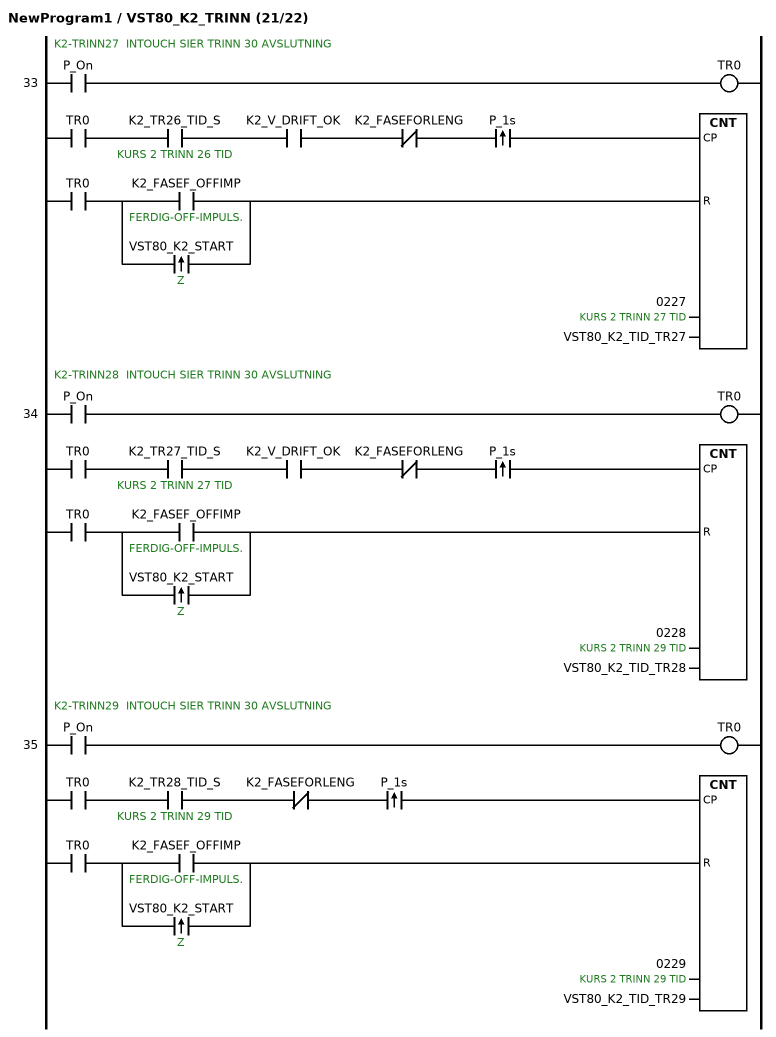
; [picture p216: NewProgram1 / VST80_K2_TRINN, rungs 33-35]
; rung 33: K2-TRINN27  INTOUCH SIER TRINN 30 AVSLUTNING
LD P_On
OUT TR0
AND K2_TR26_TID_S  ; KURS 2 TRINN 26 TID
AND K2_V_DRIFT_OK
ANDNOT K2_FASEFORLENG
@AND P_1s
LD TR0
LD K2_FASEF_OFFIMP  ; FERDIG-OFF-IMPULS.
@OR VST80_K2_START  ; Z
ANDLD
CNT 0227 VST80_K2_TID_TR27  ; KURS 2 TRINN 27 TID
; rung 34: K2-TRINN28  INTOUCH SIER TRINN 30 AVSLUTNING
LD P_On
OUT TR0
AND K2_TR27_TID_S  ; KURS 2 TRINN 27 TID
AND K2_V_DRIFT_OK
ANDNOT K2_FASEFORLENG
@AND P_1s
LD TR0
LD K2_FASEF_OFFIMP  ; FERDIG-OFF-IMPULS.
@OR VST80_K2_START  ; Z
ANDLD
CNT 0228 VST80_K2_TID_TR28  ; KURS 2 TRINN 29 TID
; rung 35: K2-TRINN29  INTOUCH SIER TRINN 30 AVSLUTNING
LD P_On
OUT TR0
AND K2_TR28_TID_S  ; KURS 2 TRINN 29 TID
ANDNOT K2_FASEFORLENG
@AND P_1s
LD TR0
LD K2_FASEF_OFFIMP  ; FERDIG-OFF-IMPULS.
@OR VST80_K2_START  ; Z
ANDLD
CNT 0229 VST80_K2_TID_TR29  ; KURS 2 TRINN 29 TID

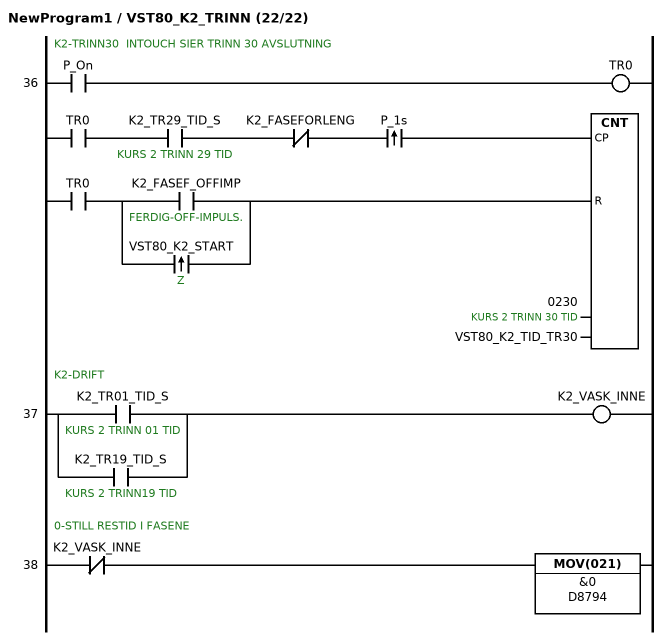
; rung 36: K2-TRINN30  INTOUCH SIER TRINN 30 AVSLUTNING
LD P_On
OUT TR0
AND K2_TR29_TID_S  ; KURS 2 TRINN 29 TID
ANDNOT K2_FASEFORLENG
@AND P_1s
LD TR0
LD K2_FASEF_OFFIMP  ; FERDIG-OFF-IMPULS.
@OR VST80_K2_START  ; Z
ANDLD
CNT 0230 VST80_K2_TID_TR30  ; KURS 2 TRINN 30 TID
; rung 37: K2-DRIFT
LD K2_TR01_TID_S  ; KURS 2 TRINN 01 TID
OR K2_TR19_TID_S  ; KURS 2 TRINN19 TID
OUT K2_VASK_INNE
; rung 38: 0-STILL RESTID I FASENE
LDNOT K2_VASK_INNE
MOV(021) &0 D8794

### Section VST80_K2_ANALOGSIGN_INN

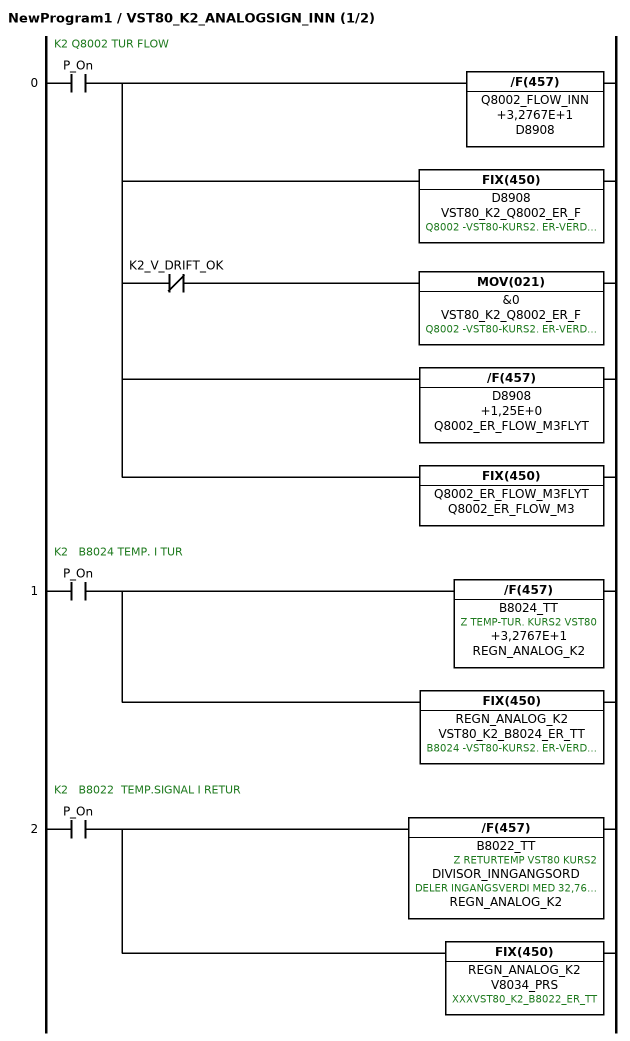
; rung 0: K2 Q8002 TUR FLOW
LD P_On
OUT TR0
/F(457) Q8002_FLOW_INN +3,2767E+1 D8908
FIX(450) D8908 VST80_K2_Q8002_ER_F  ; Q8002 -VST80-KURS2. ER-VERDI FLOW I TUR
ANDNOT K2_V_DRIFT_OK
MOV(021) &0 VST80_K2_Q8002_ER_F  ; Q8002 -VST80-KURS2. ER-VERDI FLOW I TUR
LD TR0
/F(457) D8908 +1,25E+0 Q8002_ER_FLOW_M3FLYT
FIX(450) Q8002_ER_FLOW_M3FLYT Q8002_ER_FLOW_M3
; rung 1: K2   B8024 TEMP. I TUR
LD P_On
/F(457) B8024_TT +3,2767E+1 REGN_ANALOG_K2  ; Z TEMP-TUR. KURS2 VST80
FIX(450) REGN_ANALOG_K2 VST80_K2_B8024_ER_TT  ; B8024 -VST80-KURS2. ER-VERDI TEMPERATUR I TUR TIL VST
; rung 2: K2   B8022  TEMP.SIGNAL I RETUR
LD P_On
/F(457) B8022_TT DIVISOR_INNGANGSORD REGN_ANALOG_K2  ; Z RETURTEMP VST80 KURS2, DELER INGANGSVERDI MED 32,760 FOR OMREGNING TIL 0-1000
FIX(450) REGN_ANALOG_K2 V8034_PRS  ; XXXVST80_K2_B8022_ER_TT

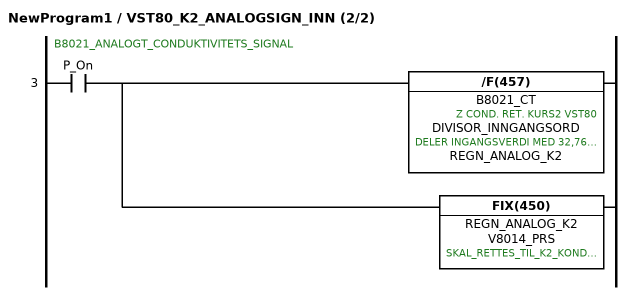
; rung 3: B8021_ANALOGT_CONDUKTIVITETS_SIGNAL
LD P_On
/F(457) B8021_CT DIVISOR_INNGANGSORD REGN_ANALOG_K2  ; Z COND. RET. KURS2 VST80, DELER INGANGSVERDI MED 32,760 FOR OMREGNING TIL 0-1000
FIX(450) REGN_ANALOG_K2 V8014_PRS  ; SKAL_RETTES_TIL_K2_KOND_ERVERDI

### Section VST_80_K2_TYPE_VASK
; KOMMANDOGIVNING FOR VALG AV TYPE VASK. / 2: DESINFEKSJON / 3: FORSKYLL

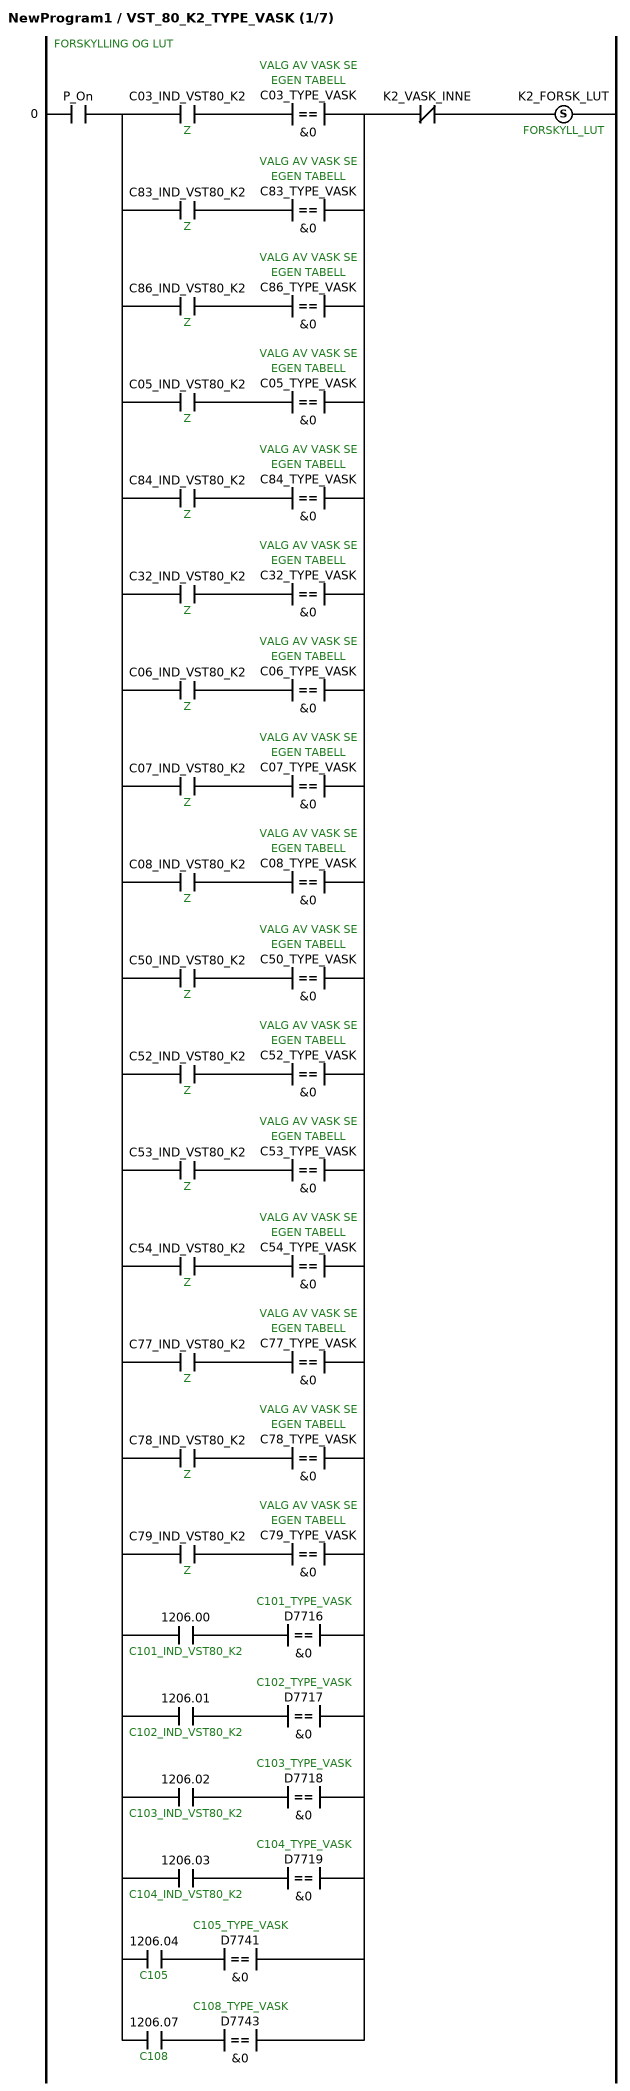
; rung 0: FORSKYLLING OG LUT
LD P_On
LD C03_IND_VST80_K2  ; Z
AND=(300) C03_TYPE_VASK &0  ; VALG AV VASK SE EGEN TABELL
LD C83_IND_VST80_K2  ; Z
AND=(300) C83_TYPE_VASK &0  ; VALG AV VASK SE EGEN TABELL
ORLD
LD C86_IND_VST80_K2  ; Z
AND=(300) C86_TYPE_VASK &0  ; VALG AV VASK SE EGEN TABELL
ORLD
LD C05_IND_VST80_K2  ; Z
AND=(300) C05_TYPE_VASK &0  ; VALG AV VASK SE EGEN TABELL
ORLD
LD C84_IND_VST80_K2  ; Z
AND=(300) C84_TYPE_VASK &0  ; VALG AV VASK SE EGEN TABELL
ORLD
LD C32_IND_VST80_K2  ; Z
AND=(300) C32_TYPE_VASK &0  ; VALG AV VASK SE EGEN TABELL
ORLD
LD C06_IND_VST80_K2  ; Z
AND=(300) C06_TYPE_VASK &0  ; VALG AV VASK SE EGEN TABELL
ORLD
LD C07_IND_VST80_K2  ; Z
AND=(300) C07_TYPE_VASK &0  ; VALG AV VASK SE EGEN TABELL
ORLD
LD C08_IND_VST80_K2  ; Z
AND=(300) C08_TYPE_VASK &0  ; VALG AV VASK SE EGEN TABELL
ORLD
LD C50_IND_VST80_K2  ; Z
AND=(300) C50_TYPE_VASK &0  ; VALG AV VASK SE EGEN TABELL
ORLD
LD C52_IND_VST80_K2  ; Z
AND=(300) C52_TYPE_VASK &0  ; VALG AV VASK SE EGEN TABELL
ORLD
LD C53_IND_VST80_K2  ; Z
AND=(300) C53_TYPE_VASK &0  ; VALG AV VASK SE EGEN TABELL
ORLD
LD C54_IND_VST80_K2  ; Z
AND=(300) C54_TYPE_VASK &0  ; VALG AV VASK SE EGEN TABELL
ORLD
LD C77_IND_VST80_K2  ; Z
AND=(300) C77_TYPE_VASK &0  ; VALG AV VASK SE EGEN TABELL
ORLD
LD C78_IND_VST80_K2  ; Z
AND=(300) C78_TYPE_VASK &0  ; VALG AV VASK SE EGEN TABELL
ORLD
LD C79_IND_VST80_K2  ; Z
AND=(300) C79_TYPE_VASK &0  ; VALG AV VASK SE EGEN TABELL
ORLD
LD 1206.00  ; C101_IND_VST80_K2
AND=(300) D7716 &0  ; C101_TYPE_VASK
ORLD
LD 1206.01  ; C102_IND_VST80_K2
AND=(300) D7717 &0  ; C102_TYPE_VASK
ORLD
LD 1206.02  ; C103_IND_VST80_K2
AND=(300) D7718 &0  ; C103_TYPE_VASK
ORLD
LD 1206.03  ; C104_IND_VST80_K2
AND=(300) D7719 &0  ; C104_TYPE_VASK
ORLD
LD 1206.04  ; C105
AND=(300) D7741 &0  ; C105_TYPE_VASK
ORLD
LD 1206.07  ; C108
AND=(300) D7743 &0  ; C108_TYPE_VASK
ORLD
ANDLD
ANDNOT K2_VASK_INNE
SET K2_FORSK_LUT  ; FORSKYLL_LUT

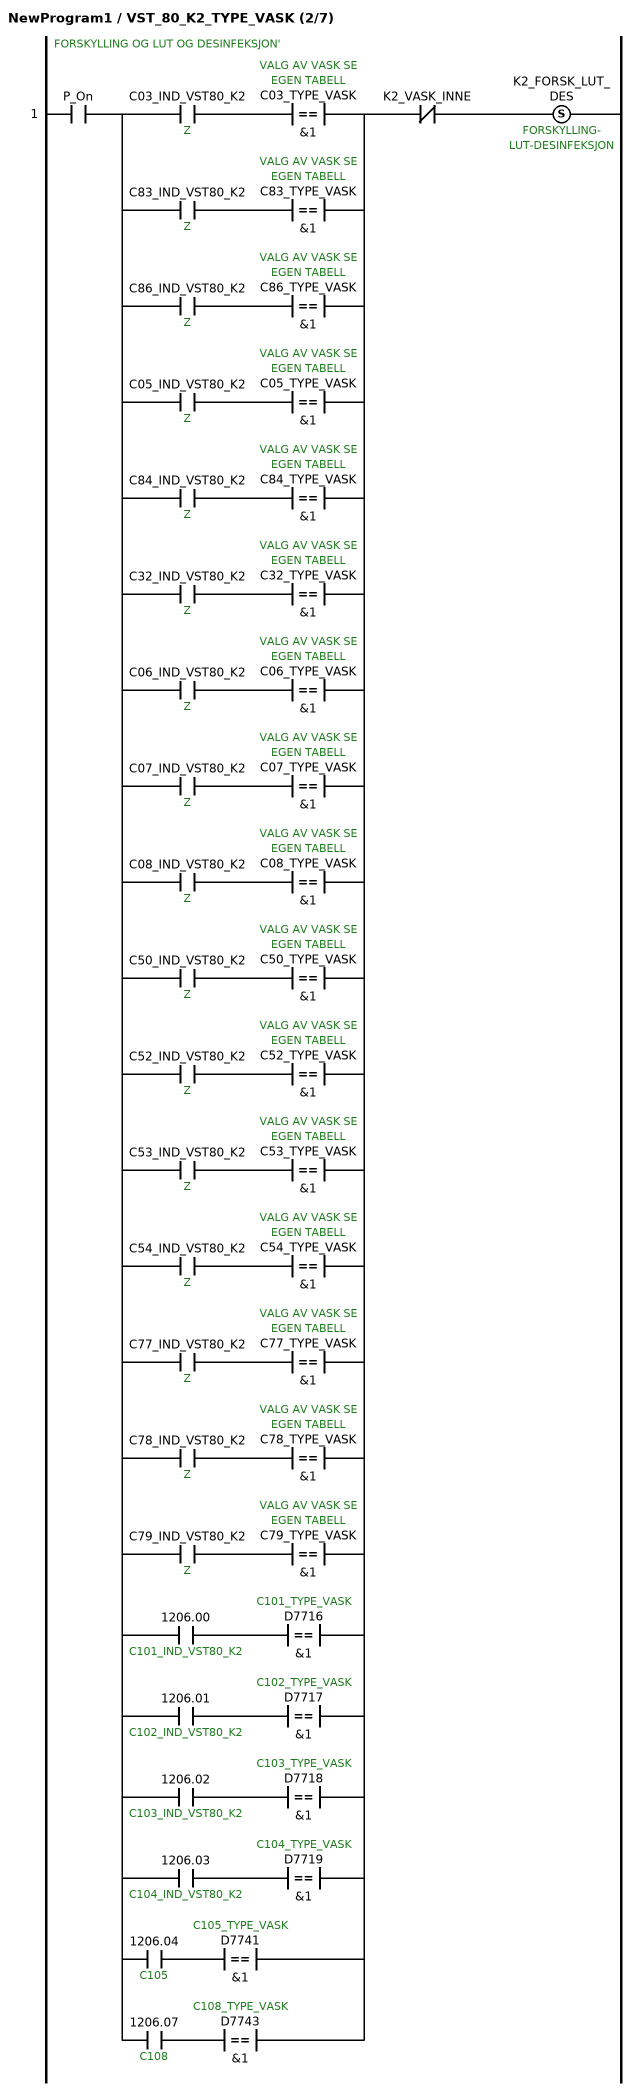
; rung 1: FORSKYLLING OG LUT OG DESINFEKSJON'
LD P_On
LD C03_IND_VST80_K2  ; Z
AND=(300) C03_TYPE_VASK &1  ; VALG AV VASK SE EGEN TABELL
LD C83_IND_VST80_K2  ; Z
AND=(300) C83_TYPE_VASK &1  ; VALG AV VASK SE EGEN TABELL
ORLD
LD C86_IND_VST80_K2  ; Z
AND=(300) C86_TYPE_VASK &1  ; VALG AV VASK SE EGEN TABELL
ORLD
LD C05_IND_VST80_K2  ; Z
AND=(300) C05_TYPE_VASK &1  ; VALG AV VASK SE EGEN TABELL
ORLD
LD C84_IND_VST80_K2  ; Z
AND=(300) C84_TYPE_VASK &1  ; VALG AV VASK SE EGEN TABELL
ORLD
LD C32_IND_VST80_K2  ; Z
AND=(300) C32_TYPE_VASK &1  ; VALG AV VASK SE EGEN TABELL
ORLD
LD C06_IND_VST80_K2  ; Z
AND=(300) C06_TYPE_VASK &1  ; VALG AV VASK SE EGEN TABELL
ORLD
LD C07_IND_VST80_K2  ; Z
AND=(300) C07_TYPE_VASK &1  ; VALG AV VASK SE EGEN TABELL
ORLD
LD C08_IND_VST80_K2  ; Z
AND=(300) C08_TYPE_VASK &1  ; VALG AV VASK SE EGEN TABELL
ORLD
LD C50_IND_VST80_K2  ; Z
AND=(300) C50_TYPE_VASK &1  ; VALG AV VASK SE EGEN TABELL
ORLD
LD C52_IND_VST80_K2  ; Z
AND=(300) C52_TYPE_VASK &1  ; VALG AV VASK SE EGEN TABELL
ORLD
LD C53_IND_VST80_K2  ; Z
AND=(300) C53_TYPE_VASK &1  ; VALG AV VASK SE EGEN TABELL
ORLD
LD C54_IND_VST80_K2  ; Z
AND=(300) C54_TYPE_VASK &1  ; VALG AV VASK SE EGEN TABELL
ORLD
LD C77_IND_VST80_K2  ; Z
AND=(300) C77_TYPE_VASK &1  ; VALG AV VASK SE EGEN TABELL
ORLD
LD C78_IND_VST80_K2  ; Z
AND=(300) C78_TYPE_VASK &1  ; VALG AV VASK SE EGEN TABELL
ORLD
LD C79_IND_VST80_K2  ; Z
AND=(300) C79_TYPE_VASK &1  ; VALG AV VASK SE EGEN TABELL
ORLD
LD 1206.00  ; C101_IND_VST80_K2
AND=(300) D7716 &1  ; C101_TYPE_VASK
ORLD
LD 1206.01  ; C102_IND_VST80_K2
AND=(300) D7717 &1  ; C102_TYPE_VASK
ORLD
LD 1206.02  ; C103_IND_VST80_K2
AND=(300) D7718 &1  ; C103_TYPE_VASK
ORLD
LD 1206.03  ; C104_IND_VST80_K2
AND=(300) D7719 &1  ; C104_TYPE_VASK
ORLD
LD 1206.04  ; C105
AND=(300) D7741 &1  ; C105_TYPE_VASK
ORLD
LD 1206.07  ; C108
AND=(300) D7743 &1  ; C108_TYPE_VASK
ORLD
ANDLD
ANDNOT K2_VASK_INNE
SET K2_FORSK_LUT_DES  ; FORSKYLLING- LUT-DESINFEKSJON

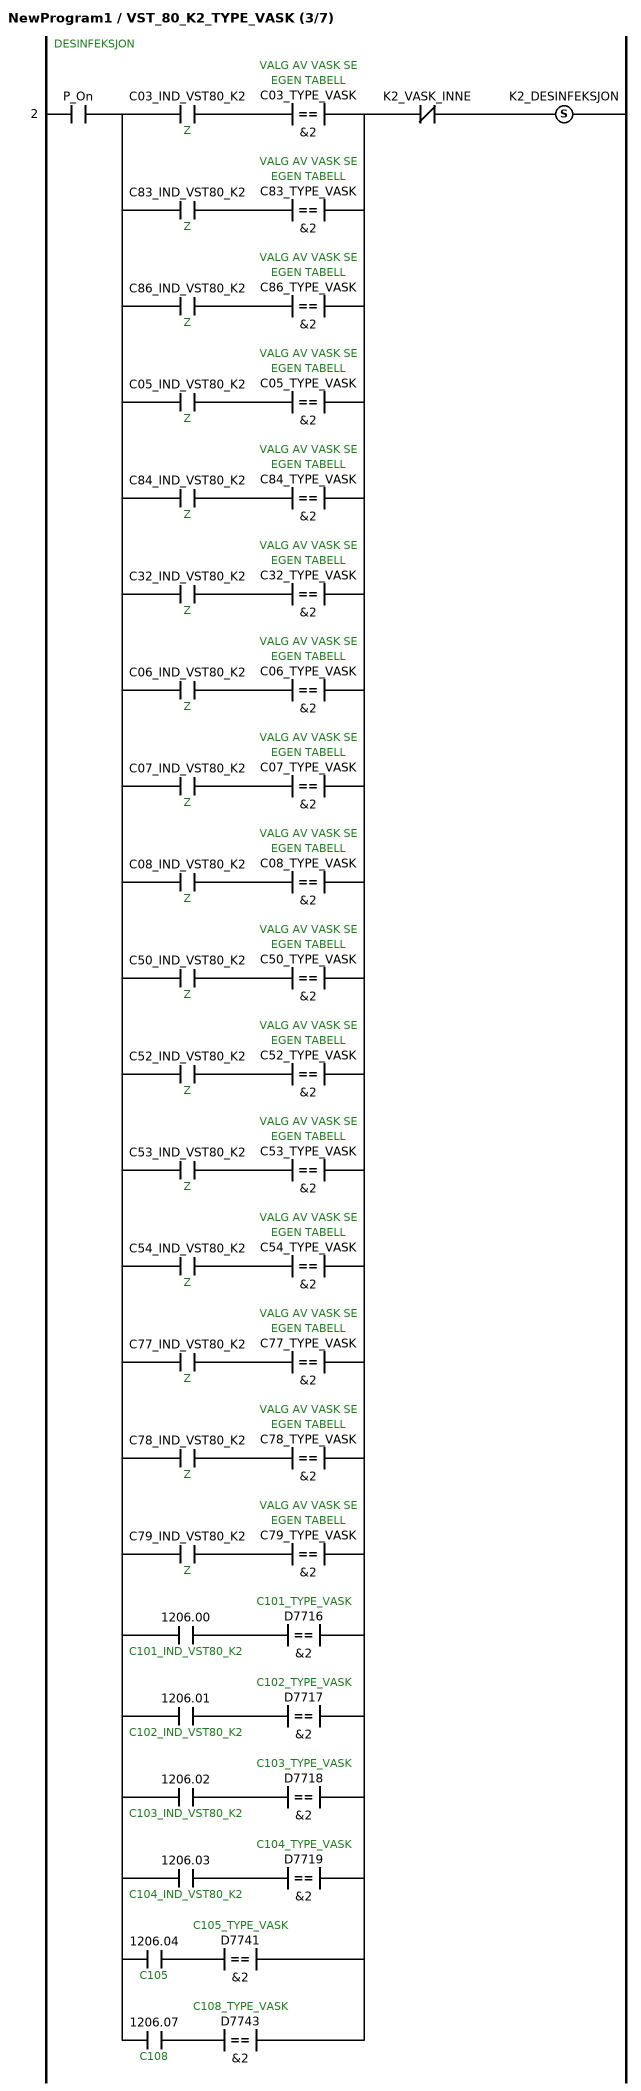
; rung 2: DESINFEKSJON
LD P_On
LD C03_IND_VST80_K2  ; Z
AND=(300) C03_TYPE_VASK &2  ; VALG AV VASK SE EGEN TABELL
LD C83_IND_VST80_K2  ; Z
AND=(300) C83_TYPE_VASK &2  ; VALG AV VASK SE EGEN TABELL
ORLD
LD C86_IND_VST80_K2  ; Z
AND=(300) C86_TYPE_VASK &2  ; VALG AV VASK SE EGEN TABELL
ORLD
LD C05_IND_VST80_K2  ; Z
AND=(300) C05_TYPE_VASK &2  ; VALG AV VASK SE EGEN TABELL
ORLD
LD C84_IND_VST80_K2  ; Z
AND=(300) C84_TYPE_VASK &2  ; VALG AV VASK SE EGEN TABELL
ORLD
LD C32_IND_VST80_K2  ; Z
AND=(300) C32_TYPE_VASK &2  ; VALG AV VASK SE EGEN TABELL
ORLD
LD C06_IND_VST80_K2  ; Z
AND=(300) C06_TYPE_VASK &2  ; VALG AV VASK SE EGEN TABELL
ORLD
LD C07_IND_VST80_K2  ; Z
AND=(300) C07_TYPE_VASK &2  ; VALG AV VASK SE EGEN TABELL
ORLD
LD C08_IND_VST80_K2  ; Z
AND=(300) C08_TYPE_VASK &2  ; VALG AV VASK SE EGEN TABELL
ORLD
LD C50_IND_VST80_K2  ; Z
AND=(300) C50_TYPE_VASK &2  ; VALG AV VASK SE EGEN TABELL
ORLD
LD C52_IND_VST80_K2  ; Z
AND=(300) C52_TYPE_VASK &2  ; VALG AV VASK SE EGEN TABELL
ORLD
LD C53_IND_VST80_K2  ; Z
AND=(300) C53_TYPE_VASK &2  ; VALG AV VASK SE EGEN TABELL
ORLD
LD C54_IND_VST80_K2  ; Z
AND=(300) C54_TYPE_VASK &2  ; VALG AV VASK SE EGEN TABELL
ORLD
LD C77_IND_VST80_K2  ; Z
AND=(300) C77_TYPE_VASK &2  ; VALG AV VASK SE EGEN TABELL
ORLD
LD C78_IND_VST80_K2  ; Z
AND=(300) C78_TYPE_VASK &2  ; VALG AV VASK SE EGEN TABELL
ORLD
LD C79_IND_VST80_K2  ; Z
AND=(300) C79_TYPE_VASK &2  ; VALG AV VASK SE EGEN TABELL
ORLD
LD 1206.00  ; C101_IND_VST80_K2
AND=(300) D7716 &2  ; C101_TYPE_VASK
ORLD
LD 1206.01  ; C102_IND_VST80_K2
AND=(300) D7717 &2  ; C102_TYPE_VASK
ORLD
LD 1206.02  ; C103_IND_VST80_K2
AND=(300) D7718 &2  ; C103_TYPE_VASK
ORLD
LD 1206.03  ; C104_IND_VST80_K2
AND=(300) D7719 &2  ; C104_TYPE_VASK
ORLD
LD 1206.04  ; C105
AND=(300) D7741 &2  ; C105_TYPE_VASK
ORLD
LD 1206.07  ; C108
AND=(300) D7743 &2  ; C108_TYPE_VASK
ORLD
ANDLD
ANDNOT K2_VASK_INNE
SET K2_DESINFEKSJON

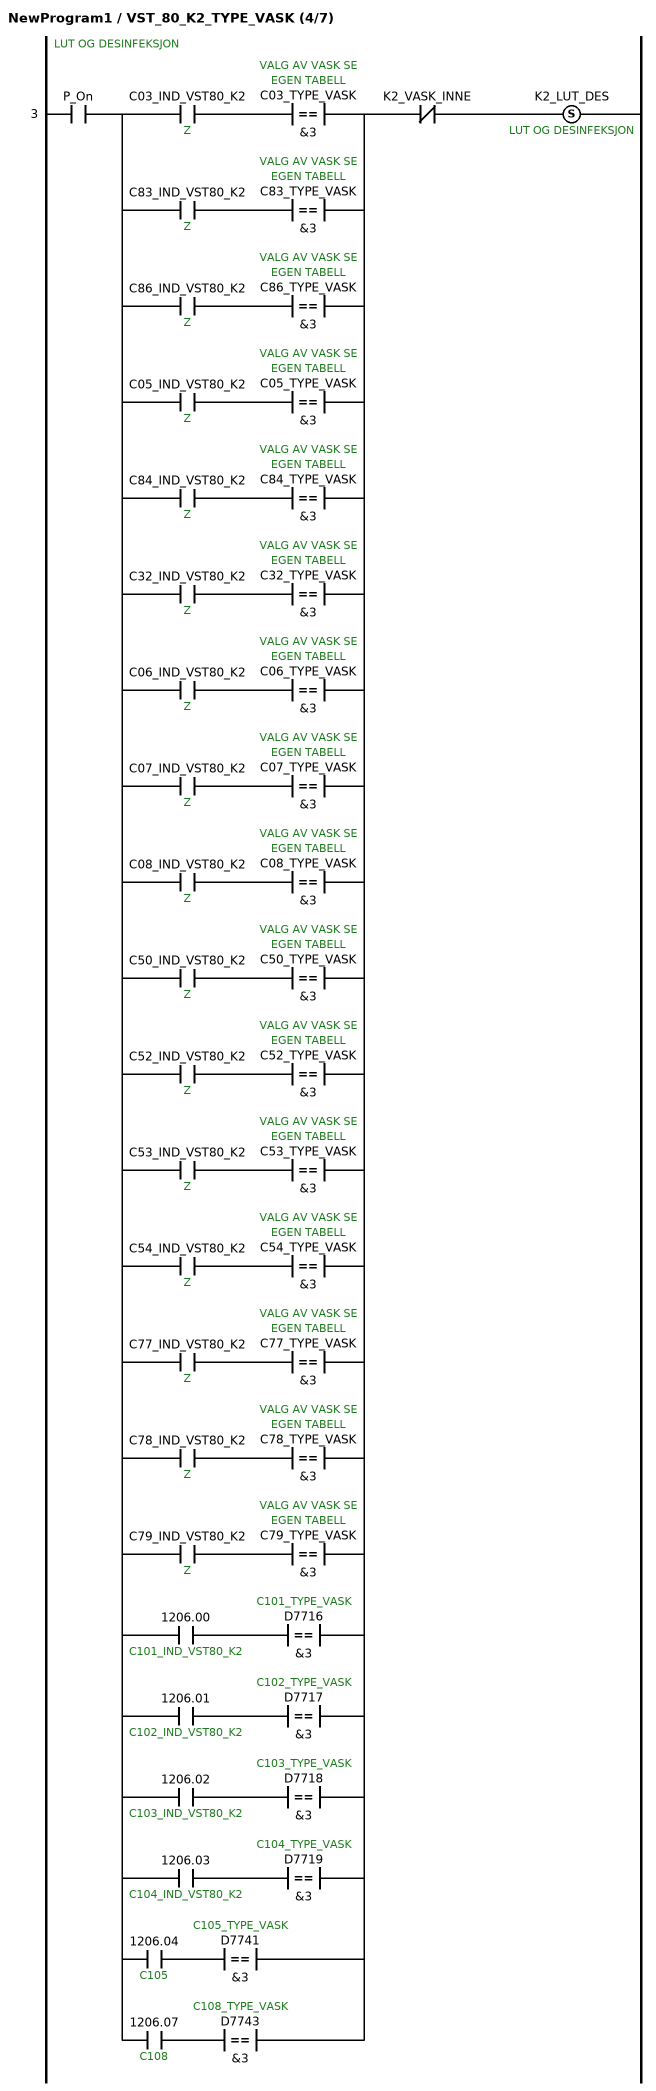
; rung 3: LUT OG DESINFEKSJON
LD P_On
LD C03_IND_VST80_K2  ; Z
AND=(300) C03_TYPE_VASK &3  ; VALG AV VASK SE EGEN TABELL
LD C83_IND_VST80_K2  ; Z
AND=(300) C83_TYPE_VASK &3  ; VALG AV VASK SE EGEN TABELL
ORLD
LD C86_IND_VST80_K2  ; Z
AND=(300) C86_TYPE_VASK &3  ; VALG AV VASK SE EGEN TABELL
ORLD
LD C05_IND_VST80_K2  ; Z
AND=(300) C05_TYPE_VASK &3  ; VALG AV VASK SE EGEN TABELL
ORLD
LD C84_IND_VST80_K2  ; Z
AND=(300) C84_TYPE_VASK &3  ; VALG AV VASK SE EGEN TABELL
ORLD
LD C32_IND_VST80_K2  ; Z
AND=(300) C32_TYPE_VASK &3  ; VALG AV VASK SE EGEN TABELL
ORLD
LD C06_IND_VST80_K2  ; Z
AND=(300) C06_TYPE_VASK &3  ; VALG AV VASK SE EGEN TABELL
ORLD
LD C07_IND_VST80_K2  ; Z
AND=(300) C07_TYPE_VASK &3  ; VALG AV VASK SE EGEN TABELL
ORLD
LD C08_IND_VST80_K2  ; Z
AND=(300) C08_TYPE_VASK &3  ; VALG AV VASK SE EGEN TABELL
ORLD
LD C50_IND_VST80_K2  ; Z
AND=(300) C50_TYPE_VASK &3  ; VALG AV VASK SE EGEN TABELL
ORLD
LD C52_IND_VST80_K2  ; Z
AND=(300) C52_TYPE_VASK &3  ; VALG AV VASK SE EGEN TABELL
ORLD
LD C53_IND_VST80_K2  ; Z
AND=(300) C53_TYPE_VASK &3  ; VALG AV VASK SE EGEN TABELL
ORLD
LD C54_IND_VST80_K2  ; Z
AND=(300) C54_TYPE_VASK &3  ; VALG AV VASK SE EGEN TABELL
ORLD
LD C77_IND_VST80_K2  ; Z
AND=(300) C77_TYPE_VASK &3  ; VALG AV VASK SE EGEN TABELL
ORLD
LD C78_IND_VST80_K2  ; Z
AND=(300) C78_TYPE_VASK &3  ; VALG AV VASK SE EGEN TABELL
ORLD
LD C79_IND_VST80_K2  ; Z
AND=(300) C79_TYPE_VASK &3  ; VALG AV VASK SE EGEN TABELL
ORLD
LD 1206.00  ; C101_IND_VST80_K2
AND=(300) D7716 &3  ; C101_TYPE_VASK
ORLD
LD 1206.01  ; C102_IND_VST80_K2
AND=(300) D7717 &3  ; C102_TYPE_VASK
ORLD
LD 1206.02  ; C103_IND_VST80_K2
AND=(300) D7718 &3  ; C103_TYPE_VASK
ORLD
LD 1206.03  ; C104_IND_VST80_K2
AND=(300) D7719 &3  ; C104_TYPE_VASK
ORLD
LD 1206.04  ; C105
AND=(300) D7741 &3  ; C105_TYPE_VASK
ORLD
LD 1206.07  ; C108
AND=(300) D7743 &3  ; C108_TYPE_VASK
ORLD
ANDLD
ANDNOT K2_VASK_INNE
SET K2_LUT_DES  ; LUT OG DESINFEKSJON

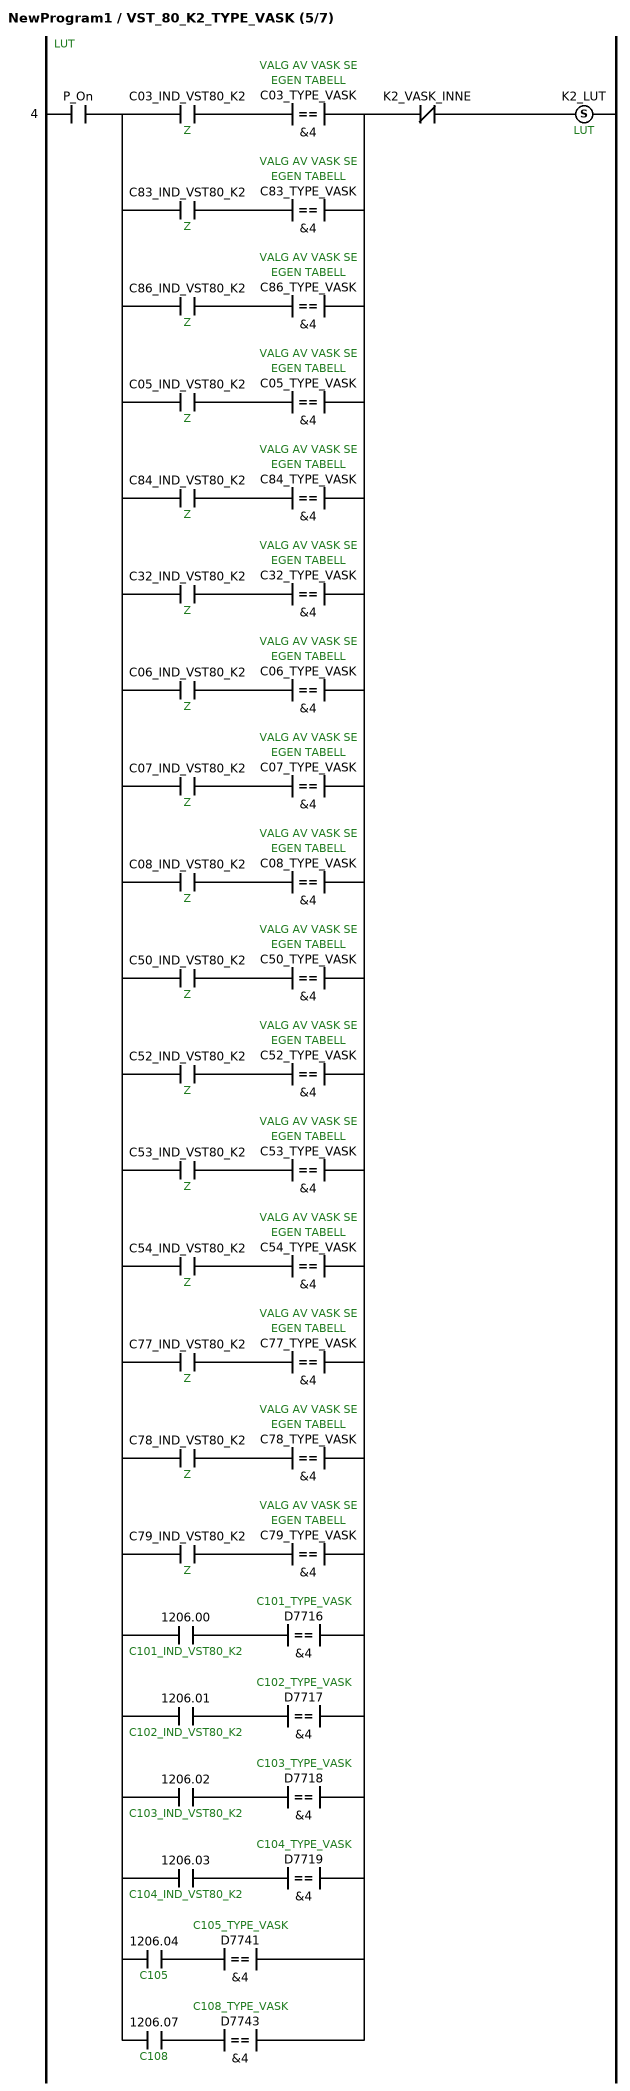
; rung 4: LUT
LD P_On
LD C03_IND_VST80_K2  ; Z
AND=(300) C03_TYPE_VASK &4  ; VALG AV VASK SE EGEN TABELL
LD C83_IND_VST80_K2  ; Z
AND=(300) C83_TYPE_VASK &4  ; VALG AV VASK SE EGEN TABELL
ORLD
LD C86_IND_VST80_K2  ; Z
AND=(300) C86_TYPE_VASK &4  ; VALG AV VASK SE EGEN TABELL
ORLD
LD C05_IND_VST80_K2  ; Z
AND=(300) C05_TYPE_VASK &4  ; VALG AV VASK SE EGEN TABELL
ORLD
LD C84_IND_VST80_K2  ; Z
AND=(300) C84_TYPE_VASK &4  ; VALG AV VASK SE EGEN TABELL
ORLD
LD C32_IND_VST80_K2  ; Z
AND=(300) C32_TYPE_VASK &4  ; VALG AV VASK SE EGEN TABELL
ORLD
LD C06_IND_VST80_K2  ; Z
AND=(300) C06_TYPE_VASK &4  ; VALG AV VASK SE EGEN TABELL
ORLD
LD C07_IND_VST80_K2  ; Z
AND=(300) C07_TYPE_VASK &4  ; VALG AV VASK SE EGEN TABELL
ORLD
LD C08_IND_VST80_K2  ; Z
AND=(300) C08_TYPE_VASK &4  ; VALG AV VASK SE EGEN TABELL
ORLD
LD C50_IND_VST80_K2  ; Z
AND=(300) C50_TYPE_VASK &4  ; VALG AV VASK SE EGEN TABELL
ORLD
LD C52_IND_VST80_K2  ; Z
AND=(300) C52_TYPE_VASK &4  ; VALG AV VASK SE EGEN TABELL
ORLD
LD C53_IND_VST80_K2  ; Z
AND=(300) C53_TYPE_VASK &4  ; VALG AV VASK SE EGEN TABELL
ORLD
LD C54_IND_VST80_K2  ; Z
AND=(300) C54_TYPE_VASK &4  ; VALG AV VASK SE EGEN TABELL
ORLD
LD C77_IND_VST80_K2  ; Z
AND=(300) C77_TYPE_VASK &4  ; VALG AV VASK SE EGEN TABELL
ORLD
LD C78_IND_VST80_K2  ; Z
AND=(300) C78_TYPE_VASK &4  ; VALG AV VASK SE EGEN TABELL
ORLD
LD C79_IND_VST80_K2  ; Z
AND=(300) C79_TYPE_VASK &4  ; VALG AV VASK SE EGEN TABELL
ORLD
LD 1206.00  ; C101_IND_VST80_K2
AND=(300) D7716 &4  ; C101_TYPE_VASK
ORLD
LD 1206.01  ; C102_IND_VST80_K2
AND=(300) D7717 &4  ; C102_TYPE_VASK
ORLD
LD 1206.02  ; C103_IND_VST80_K2
AND=(300) D7718 &4  ; C103_TYPE_VASK
ORLD
LD 1206.03  ; C104_IND_VST80_K2
AND=(300) D7719 &4  ; C104_TYPE_VASK
ORLD
LD 1206.04  ; C105
AND=(300) D7741 &4  ; C105_TYPE_VASK
ORLD
LD 1206.07  ; C108
AND=(300) D7743 &4  ; C108_TYPE_VASK
ORLD
ANDLD
ANDNOT K2_VASK_INNE
SET K2_LUT  ; LUT

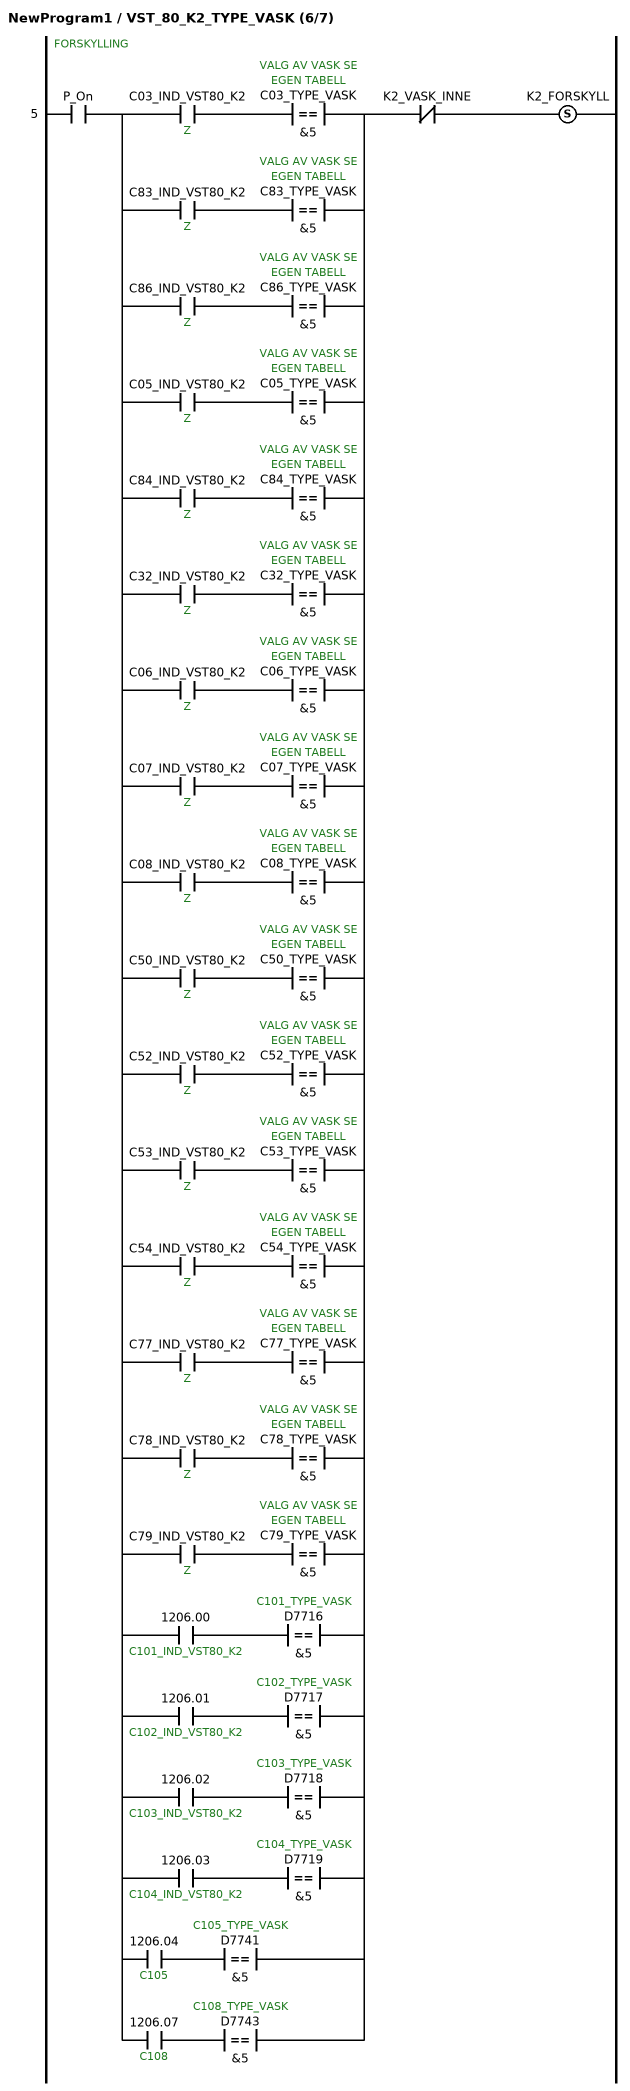
; rung 5: FORSKYLLING
LD P_On
LD C03_IND_VST80_K2  ; Z
AND=(300) C03_TYPE_VASK &5  ; VALG AV VASK SE EGEN TABELL
LD C83_IND_VST80_K2  ; Z
AND=(300) C83_TYPE_VASK &5  ; VALG AV VASK SE EGEN TABELL
ORLD
LD C86_IND_VST80_K2  ; Z
AND=(300) C86_TYPE_VASK &5  ; VALG AV VASK SE EGEN TABELL
ORLD
LD C05_IND_VST80_K2  ; Z
AND=(300) C05_TYPE_VASK &5  ; VALG AV VASK SE EGEN TABELL
ORLD
LD C84_IND_VST80_K2  ; Z
AND=(300) C84_TYPE_VASK &5  ; VALG AV VASK SE EGEN TABELL
ORLD
LD C32_IND_VST80_K2  ; Z
AND=(300) C32_TYPE_VASK &5  ; VALG AV VASK SE EGEN TABELL
ORLD
LD C06_IND_VST80_K2  ; Z
AND=(300) C06_TYPE_VASK &5  ; VALG AV VASK SE EGEN TABELL
ORLD
LD C07_IND_VST80_K2  ; Z
AND=(300) C07_TYPE_VASK &5  ; VALG AV VASK SE EGEN TABELL
ORLD
LD C08_IND_VST80_K2  ; Z
AND=(300) C08_TYPE_VASK &5  ; VALG AV VASK SE EGEN TABELL
ORLD
LD C50_IND_VST80_K2  ; Z
AND=(300) C50_TYPE_VASK &5  ; VALG AV VASK SE EGEN TABELL
ORLD
LD C52_IND_VST80_K2  ; Z
AND=(300) C52_TYPE_VASK &5  ; VALG AV VASK SE EGEN TABELL
ORLD
LD C53_IND_VST80_K2  ; Z
AND=(300) C53_TYPE_VASK &5  ; VALG AV VASK SE EGEN TABELL
ORLD
LD C54_IND_VST80_K2  ; Z
AND=(300) C54_TYPE_VASK &5  ; VALG AV VASK SE EGEN TABELL
ORLD
LD C77_IND_VST80_K2  ; Z
AND=(300) C77_TYPE_VASK &5  ; VALG AV VASK SE EGEN TABELL
ORLD
LD C78_IND_VST80_K2  ; Z
AND=(300) C78_TYPE_VASK &5  ; VALG AV VASK SE EGEN TABELL
ORLD
LD C79_IND_VST80_K2  ; Z
AND=(300) C79_TYPE_VASK &5  ; VALG AV VASK SE EGEN TABELL
ORLD
LD 1206.00  ; C101_IND_VST80_K2
AND=(300) D7716 &5  ; C101_TYPE_VASK
ORLD
LD 1206.01  ; C102_IND_VST80_K2
AND=(300) D7717 &5  ; C102_TYPE_VASK
ORLD
LD 1206.02  ; C103_IND_VST80_K2
AND=(300) D7718 &5  ; C103_TYPE_VASK
ORLD
LD 1206.03  ; C104_IND_VST80_K2
AND=(300) D7719 &5  ; C104_TYPE_VASK
ORLD
LD 1206.04  ; C105
AND=(300) D7741 &5  ; C105_TYPE_VASK
ORLD
LD 1206.07  ; C108
AND=(300) D7743 &5  ; C108_TYPE_VASK
ORLD
ANDLD
ANDNOT K2_VASK_INNE
SET K2_FORSKYLL

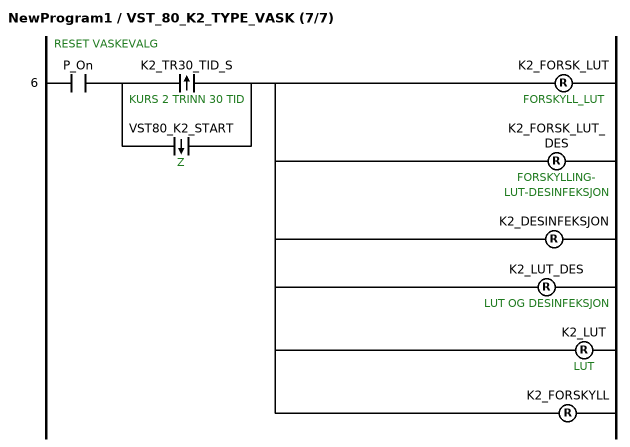
; rung 6: RESET VASKEVALG
LD P_On
@LD K2_TR30_TID_S  ; KURS 2 TRINN 30 TID
%OR VST80_K2_START  ; Z
ANDLD
RSET K2_FORSK_LUT  ; FORSKYLL_LUT
RSET K2_FORSK_LUT_DES  ; FORSKYLLING- LUT-DESINFEKSJON
RSET K2_DESINFEKSJON
RSET K2_LUT_DES  ; LUT OG DESINFEKSJON
RSET K2_LUT  ; LUT
RSET K2_FORSKYLL

### Section VST80_K2_DR_STATUS

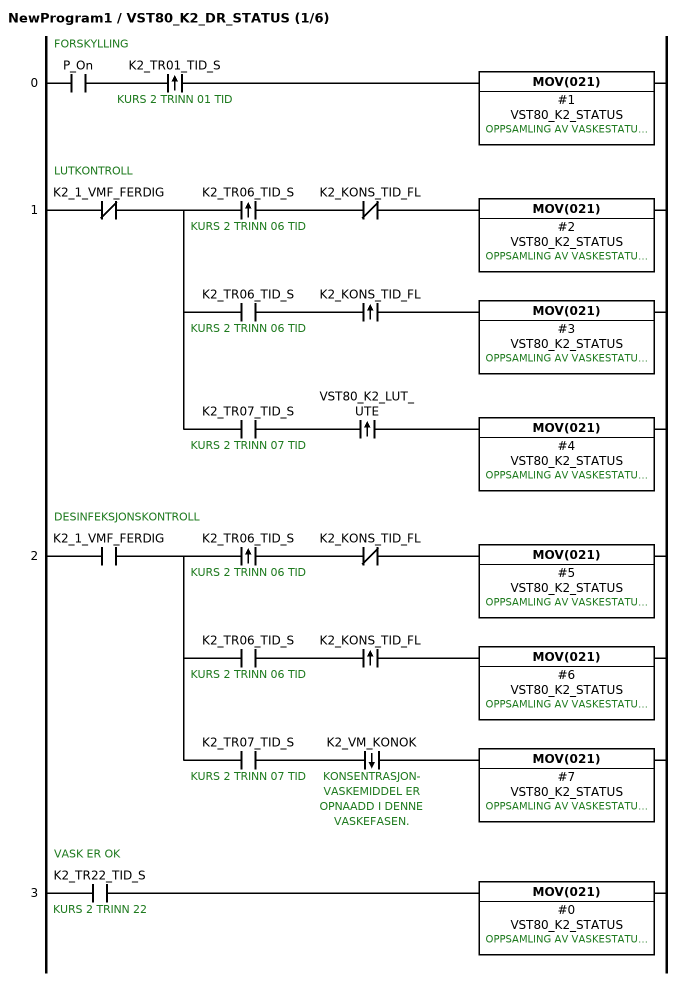
; rung 0: FORSKYLLING
LD P_On
@AND K2_TR01_TID_S  ; KURS 2 TRINN 01 TID
MOV(021) #1 VST80_K2_STATUS  ; OPPSAMLING AV VASKESTATUS UNDER VASK
; rung 1: LUTKONTROLL
LDNOT K2_1_VMF_FERDIG
OUT TR0
@AND K2_TR06_TID_S  ; KURS 2 TRINN 06 TID
ANDNOT K2_KONS_TID_FL
MOV(021) #2 VST80_K2_STATUS  ; OPPSAMLING AV VASKESTATUS UNDER VASK
LD TR0
AND K2_TR06_TID_S  ; KURS 2 TRINN 06 TID
@AND K2_KONS_TID_FL
MOV(021) #3 VST80_K2_STATUS  ; OPPSAMLING AV VASKESTATUS UNDER VASK
LD TR0
AND K2_TR07_TID_S  ; KURS 2 TRINN 07 TID
@AND VST80_K2_LUT_UTE
MOV(021) #4 VST80_K2_STATUS  ; OPPSAMLING AV VASKESTATUS UNDER VASK
; rung 2: DESINFEKSJONSKONTROLL
LD K2_1_VMF_FERDIG
OUT TR0
@AND K2_TR06_TID_S  ; KURS 2 TRINN 06 TID
ANDNOT K2_KONS_TID_FL
MOV(021) #5 VST80_K2_STATUS  ; OPPSAMLING AV VASKESTATUS UNDER VASK
LD TR0
AND K2_TR06_TID_S  ; KURS 2 TRINN 06 TID
@AND K2_KONS_TID_FL
MOV(021) #6 VST80_K2_STATUS  ; OPPSAMLING AV VASKESTATUS UNDER VASK
LD TR0
AND K2_TR07_TID_S  ; KURS 2 TRINN 07 TID
%AND K2_VM_KONOK  ; KONSENTRASJON-VASKEMIDDEL ER OPNAADD I DENNE VASKEFASEN.
MOV(021) #7 VST80_K2_STATUS  ; OPPSAMLING AV VASKESTATUS UNDER VASK
; rung 3: VASK ER OK
LD K2_TR22_TID_S  ; KURS 2 TRINN 22
MOV(021) #0 VST80_K2_STATUS  ; OPPSAMLING AV VASKESTATUS UNDER VASK

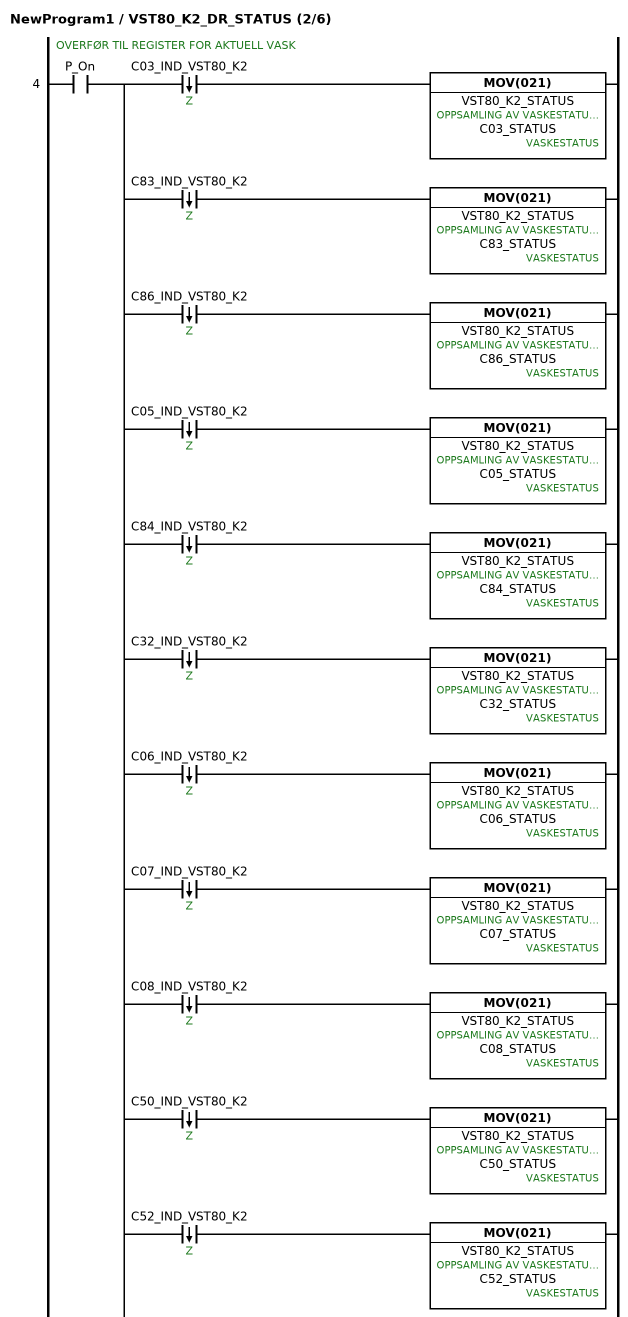

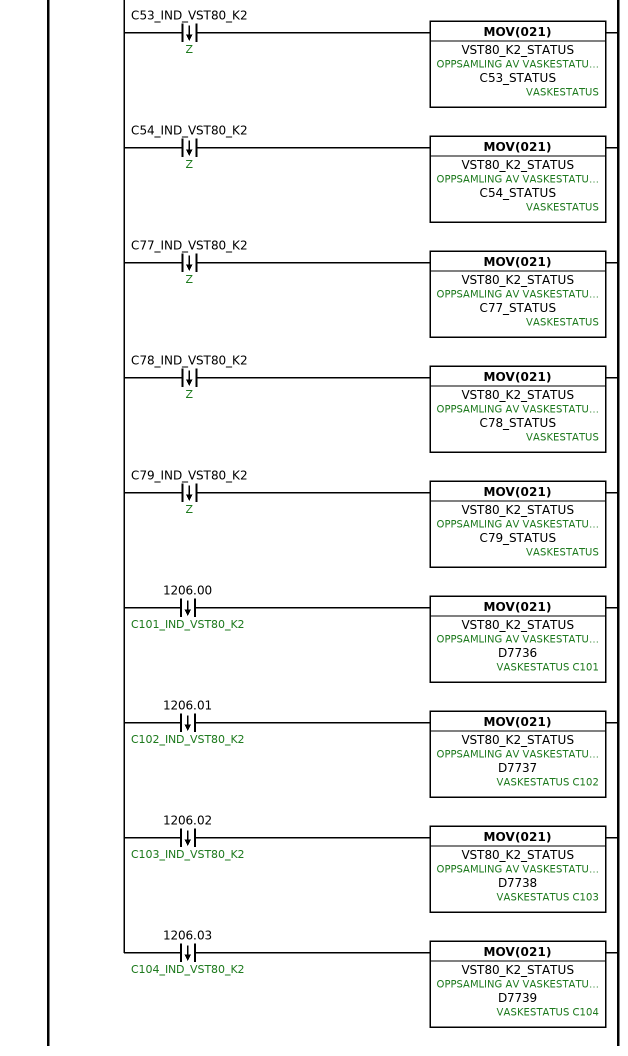
; rung 4: OVERFØR TIL REGISTER FOR AKTUELL VASK
LD P_On
OUT TR0
%AND C03_IND_VST80_K2  ; Z
MOV(021) VST80_K2_STATUS C03_STATUS  ; OPPSAMLING AV VASKESTATUS UNDER VASK, VASKESTATUS
LD TR0
%AND C83_IND_VST80_K2  ; Z
MOV(021) VST80_K2_STATUS C83_STATUS  ; OPPSAMLING AV VASKESTATUS UNDER VASK, VASKESTATUS
LD TR0
%AND C86_IND_VST80_K2  ; Z
MOV(021) VST80_K2_STATUS C86_STATUS  ; OPPSAMLING AV VASKESTATUS UNDER VASK, VASKESTATUS
LD TR0
%AND C05_IND_VST80_K2  ; Z
MOV(021) VST80_K2_STATUS C05_STATUS  ; OPPSAMLING AV VASKESTATUS UNDER VASK, VASKESTATUS
LD TR0
%AND C84_IND_VST80_K2  ; Z
MOV(021) VST80_K2_STATUS C84_STATUS  ; OPPSAMLING AV VASKESTATUS UNDER VASK, VASKESTATUS
LD TR0
%AND C32_IND_VST80_K2  ; Z
MOV(021) VST80_K2_STATUS C32_STATUS  ; OPPSAMLING AV VASKESTATUS UNDER VASK, VASKESTATUS
LD TR0
%AND C06_IND_VST80_K2  ; Z
MOV(021) VST80_K2_STATUS C06_STATUS  ; OPPSAMLING AV VASKESTATUS UNDER VASK, VASKESTATUS
LD TR0
%AND C07_IND_VST80_K2  ; Z
MOV(021) VST80_K2_STATUS C07_STATUS  ; OPPSAMLING AV VASKESTATUS UNDER VASK, VASKESTATUS
LD TR0
%AND C08_IND_VST80_K2  ; Z
MOV(021) VST80_K2_STATUS C08_STATUS  ; OPPSAMLING AV VASKESTATUS UNDER VASK, VASKESTATUS
LD TR0
%AND C50_IND_VST80_K2  ; Z
MOV(021) VST80_K2_STATUS C50_STATUS  ; OPPSAMLING AV VASKESTATUS UNDER VASK, VASKESTATUS
LD TR0
%AND C52_IND_VST80_K2  ; Z
MOV(021) VST80_K2_STATUS C52_STATUS  ; OPPSAMLING AV VASKESTATUS UNDER VASK, VASKESTATUS
LD TR0
%AND C53_IND_VST80_K2  ; Z
MOV(021) VST80_K2_STATUS C53_STATUS  ; OPPSAMLING AV VASKESTATUS UNDER VASK, VASKESTATUS
LD TR0
%AND C54_IND_VST80_K2  ; Z
MOV(021) VST80_K2_STATUS C54_STATUS  ; OPPSAMLING AV VASKESTATUS UNDER VASK, VASKESTATUS
LD TR0
%AND C77_IND_VST80_K2  ; Z
MOV(021) VST80_K2_STATUS C77_STATUS  ; OPPSAMLING AV VASKESTATUS UNDER VASK, VASKESTATUS
LD TR0
%AND C78_IND_VST80_K2  ; Z
MOV(021) VST80_K2_STATUS C78_STATUS  ; OPPSAMLING AV VASKESTATUS UNDER VASK, VASKESTATUS
LD TR0
%AND C79_IND_VST80_K2  ; Z
MOV(021) VST80_K2_STATUS C79_STATUS  ; OPPSAMLING AV VASKESTATUS UNDER VASK, VASKESTATUS
LD TR0
%AND 1206.00  ; C101_IND_VST80_K2
MOV(021) VST80_K2_STATUS D7736  ; OPPSAMLING AV VASKESTATUS UNDER VASK, VASKESTATUS C101
LD TR0
%AND 1206.01  ; C102_IND_VST80_K2
MOV(021) VST80_K2_STATUS D7737  ; OPPSAMLING AV VASKESTATUS UNDER VASK, VASKESTATUS C102
LD TR0
%AND 1206.02  ; C103_IND_VST80_K2
MOV(021) VST80_K2_STATUS D7738  ; OPPSAMLING AV VASKESTATUS UNDER VASK, VASKESTATUS C103
LD TR0
%AND 1206.03  ; C104_IND_VST80_K2
MOV(021) VST80_K2_STATUS D7739  ; OPPSAMLING AV VASKESTATUS UNDER VASK, VASKESTATUS C104

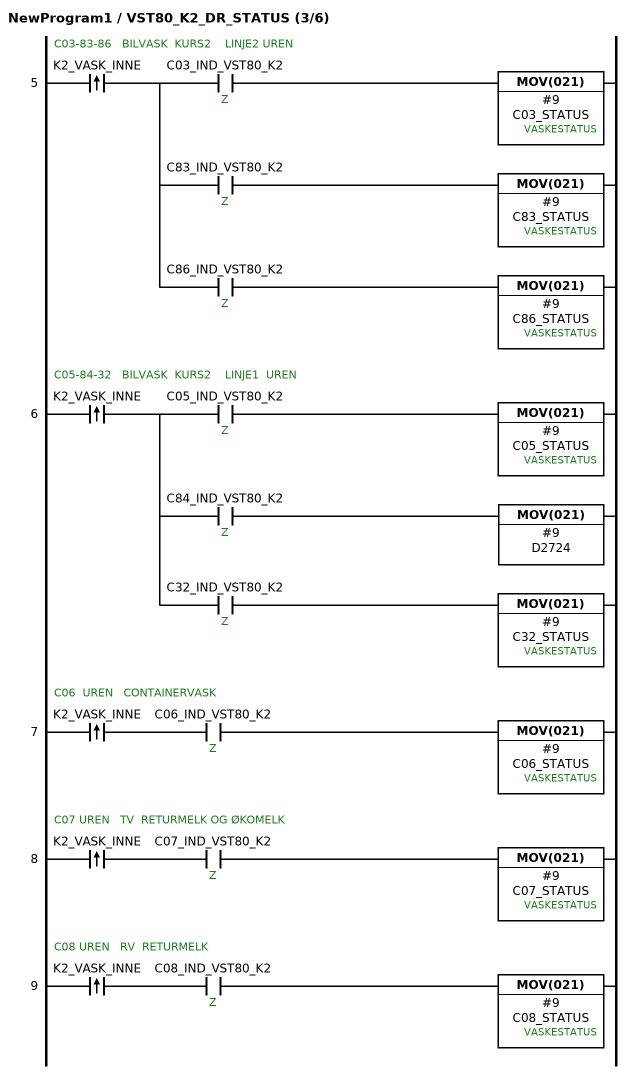
; rung 5: C03-83-86   BILVASK  KURS2    LINJE2 UREN
@LD K2_VASK_INNE
OUT TR0
AND C03_IND_VST80_K2  ; Z
MOV(021) #9 C03_STATUS  ; VASKESTATUS
LD TR0
AND C83_IND_VST80_K2  ; Z
MOV(021) #9 C83_STATUS  ; VASKESTATUS
LD TR0
AND C86_IND_VST80_K2  ; Z
MOV(021) #9 C86_STATUS  ; VASKESTATUS
; rung 6: C05-84-32   BILVASK  KURS2    LINJE1  UREN
@LD K2_VASK_INNE
OUT TR0
AND C05_IND_VST80_K2  ; Z
MOV(021) #9 C05_STATUS  ; VASKESTATUS
LD TR0
AND C84_IND_VST80_K2  ; Z
MOV(021) #9 D2724
LD TR0
AND C32_IND_VST80_K2  ; Z
MOV(021) #9 C32_STATUS  ; VASKESTATUS
; rung 7: C06  UREN   CONTAINERVASK
@LD K2_VASK_INNE
AND C06_IND_VST80_K2  ; Z
MOV(021) #9 C06_STATUS  ; VASKESTATUS
; rung 8: C07 UREN   TV  RETURMELK OG ØKOMELK
@LD K2_VASK_INNE
AND C07_IND_VST80_K2  ; Z
MOV(021) #9 C07_STATUS  ; VASKESTATUS
; rung 9: C08 UREN   RV  RETURMELK
@LD K2_VASK_INNE
AND C08_IND_VST80_K2  ; Z
MOV(021) #9 C08_STATUS  ; VASKESTATUS

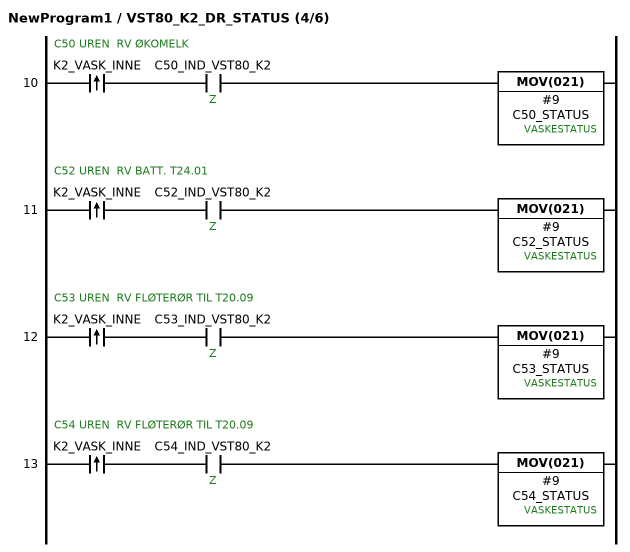
; rung 10: C50 UREN  RV ØKOMELK
@LD K2_VASK_INNE
AND C50_IND_VST80_K2  ; Z
MOV(021) #9 C50_STATUS  ; VASKESTATUS
; rung 11: C52 UREN  RV BATT. T24.01
@LD K2_VASK_INNE
AND C52_IND_VST80_K2  ; Z
MOV(021) #9 C52_STATUS  ; VASKESTATUS
; rung 12: C53 UREN  RV FLØTERØR TIL T20.09
@LD K2_VASK_INNE
AND C53_IND_VST80_K2  ; Z
MOV(021) #9 C53_STATUS  ; VASKESTATUS
; rung 13: C54 UREN  RV FLØTERØR TIL T20.09
@LD K2_VASK_INNE
AND C54_IND_VST80_K2  ; Z
MOV(021) #9 C54_STATUS  ; VASKESTATUS

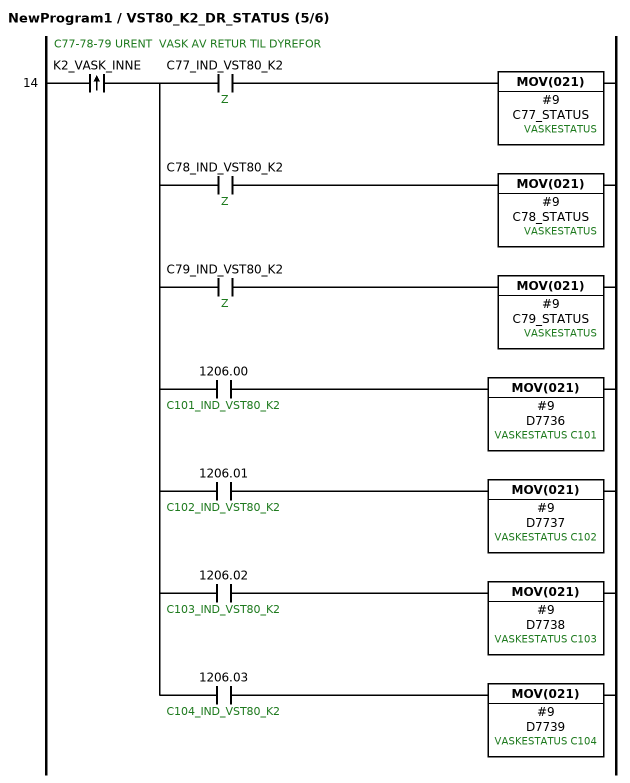
; rung 14: C77-78-79 URENT  VASK AV RETUR TIL DYREFOR
@LD K2_VASK_INNE
OUT TR0
AND C77_IND_VST80_K2  ; Z
MOV(021) #9 C77_STATUS  ; VASKESTATUS
LD TR0
AND C78_IND_VST80_K2  ; Z
MOV(021) #9 C78_STATUS  ; VASKESTATUS
LD TR0
AND C79_IND_VST80_K2  ; Z
MOV(021) #9 C79_STATUS  ; VASKESTATUS
LD TR0
AND 1206.00  ; C101_IND_VST80_K2
MOV(021) #9 D7736  ; VASKESTATUS C101
LD TR0
AND 1206.01  ; C102_IND_VST80_K2
MOV(021) #9 D7737  ; VASKESTATUS C102
LD TR0
AND 1206.02  ; C103_IND_VST80_K2
MOV(021) #9 D7738  ; VASKESTATUS C103
LD TR0
AND 1206.03  ; C104_IND_VST80_K2
MOV(021) #9 D7739  ; VASKESTATUS C104

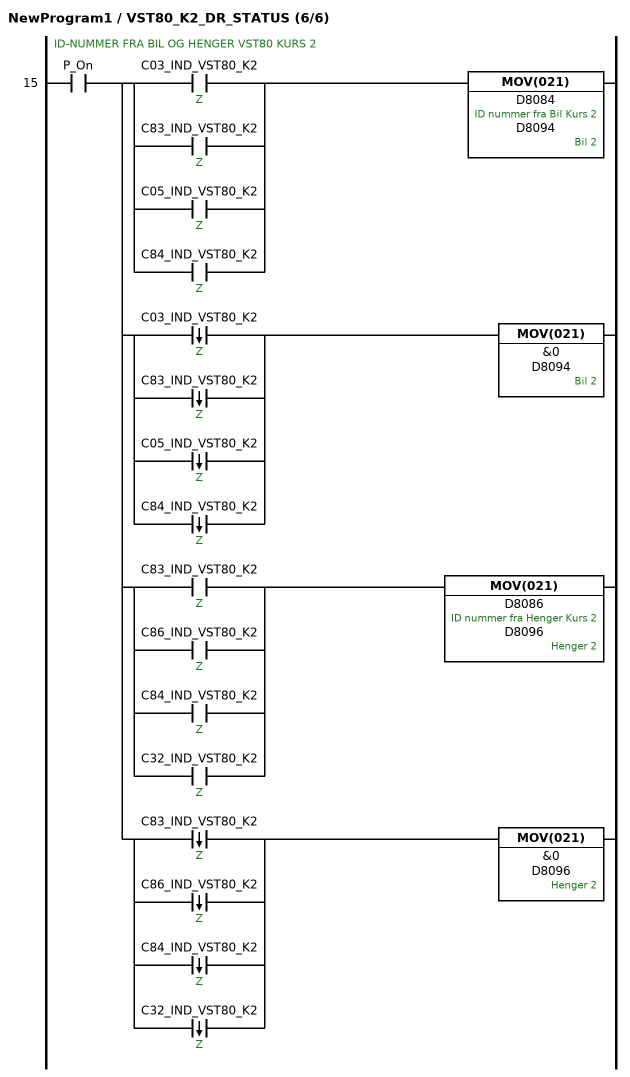
; rung 15: ID-NUMMER FRA BIL OG HENGER VST80 KURS 2
LD P_On
OUT TR0
LD C03_IND_VST80_K2  ; Z
OR C83_IND_VST80_K2  ; Z
OR C05_IND_VST80_K2  ; Z
OR C84_IND_VST80_K2  ; Z
ANDLD
MOV(021) D8084 D8094  ; ID nummer fra Bil Kurs 2, Bil 2
LD TR0
%LD C03_IND_VST80_K2  ; Z
%OR C83_IND_VST80_K2  ; Z
%OR C05_IND_VST80_K2  ; Z
%OR C84_IND_VST80_K2  ; Z
ANDLD
MOV(021) &0 D8094  ; Bil 2
LD TR0
LD C83_IND_VST80_K2  ; Z
OR C86_IND_VST80_K2  ; Z
OR C84_IND_VST80_K2  ; Z
OR C32_IND_VST80_K2  ; Z
ANDLD
MOV(021) D8086 D8096  ; ID nummer fra Henger Kurs 2, Henger 2
LD TR0
%LD C83_IND_VST80_K2  ; Z
%OR C86_IND_VST80_K2  ; Z
%OR C84_IND_VST80_K2  ; Z
%OR C32_IND_VST80_K2  ; Z
ANDLD
MOV(021) &0 D8096  ; Henger 2

### Section VST80_K2_FUNKSJON
; Dette programmet styrer kommandoene til vaskestasjonen.

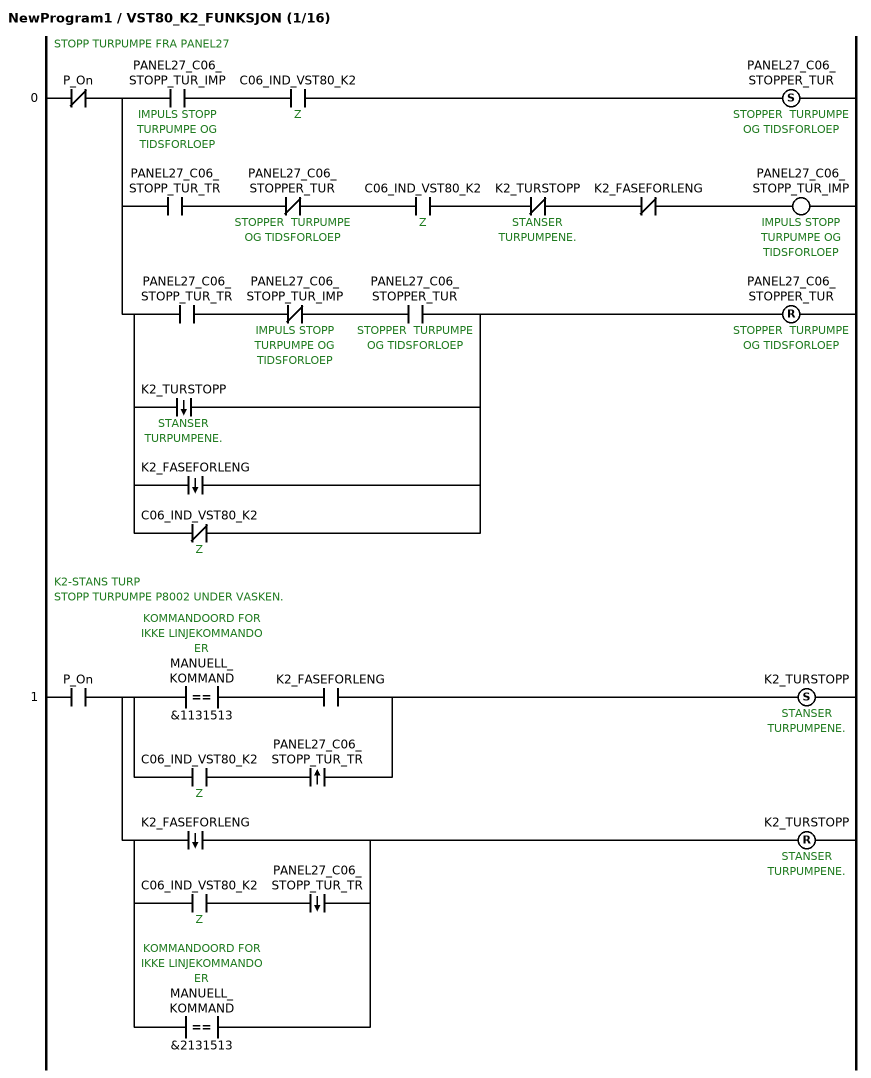
; rung 0: STOPP TURPUMPE FRA PANEL27
LDNOT P_On
OUT TR0
AND PANEL27_C06_STOPP_TUR_IMP  ; IMPULS STOPP  TURPUMPE OG TIDSFORLOEP
AND C06_IND_VST80_K2  ; Z
SET PANEL27_C06_STOPPER_TUR  ; STOPPER  TURPUMPE OG TIDSFORLOEP
LD TR0
AND PANEL27_C06_STOPP_TUR_TR
ANDNOT PANEL27_C06_STOPPER_TUR  ; STOPPER  TURPUMPE OG TIDSFORLOEP
AND C06_IND_VST80_K2  ; Z
ANDNOT K2_TURSTOPP  ; STANSER TURPUMPENE.
ANDNOT K2_FASEFORLENG
OUT PANEL27_C06_STOPP_TUR_IMP  ; IMPULS STOPP  TURPUMPE OG TIDSFORLOEP
LD TR0
LD PANEL27_C06_STOPP_TUR_TR
ANDNOT PANEL27_C06_STOPP_TUR_IMP  ; IMPULS STOPP  TURPUMPE OG TIDSFORLOEP
AND PANEL27_C06_STOPPER_TUR  ; STOPPER  TURPUMPE OG TIDSFORLOEP
%OR K2_TURSTOPP  ; STANSER TURPUMPENE.
%OR K2_FASEFORLENG
ORNOT C06_IND_VST80_K2  ; Z
ANDLD
RSET PANEL27_C06_STOPPER_TUR  ; STOPPER  TURPUMPE OG TIDSFORLOEP
; rung 1: K2-STANS TURP / STOPP TURPUMPE P8002 UNDER VASKEN.
LD P_On
OUT TR0
LD=L(301) MANUELL_KOMMAND &1131513  ; KOMMANDOORD FOR IKKE LINJEKOMMANDOER
AND K2_FASEFORLENG
LD C06_IND_VST80_K2  ; Z
@AND PANEL27_C06_STOPP_TUR_TR
ORLD
ANDLD
SET K2_TURSTOPP  ; STANSER TURPUMPENE.
LD TR0
%LD K2_FASEFORLENG
LD C06_IND_VST80_K2  ; Z
%AND PANEL27_C06_STOPP_TUR_TR
ORLD
OR=L(301) MANUELL_KOMMAND &2131513  ; KOMMANDOORD FOR IKKE LINJEKOMMANDOER
ANDLD
RSET K2_TURSTOPP  ; STANSER TURPUMPENE.

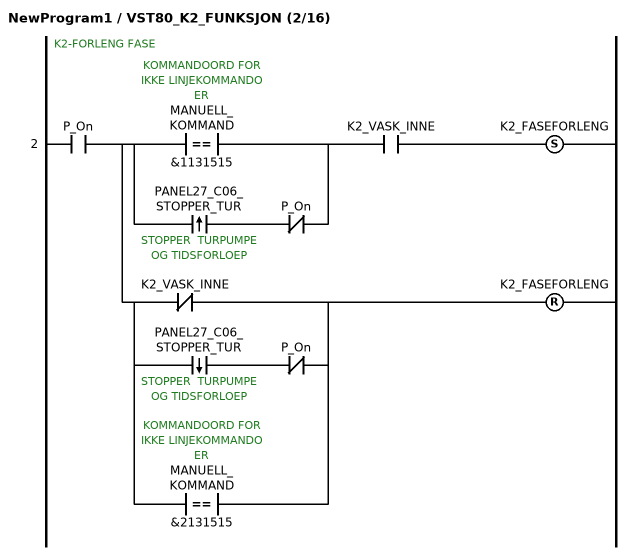
; rung 2: K2-FORLENG FASE
LD P_On
OUT TR0
LD=L(301) MANUELL_KOMMAND &1131515  ; KOMMANDOORD FOR IKKE LINJEKOMMANDOER
@LD PANEL27_C06_STOPPER_TUR  ; STOPPER  TURPUMPE OG TIDSFORLOEP
ANDNOT P_On
ORLD
ANDLD
AND K2_VASK_INNE
SET K2_FASEFORLENG
LD TR0
LDNOT K2_VASK_INNE
%LD PANEL27_C06_STOPPER_TUR  ; STOPPER  TURPUMPE OG TIDSFORLOEP
ANDNOT P_On
ORLD
OR=L(301) MANUELL_KOMMAND &2131515  ; KOMMANDOORD FOR IKKE LINJEKOMMANDOER
ANDLD
RSET K2_FASEFORLENG

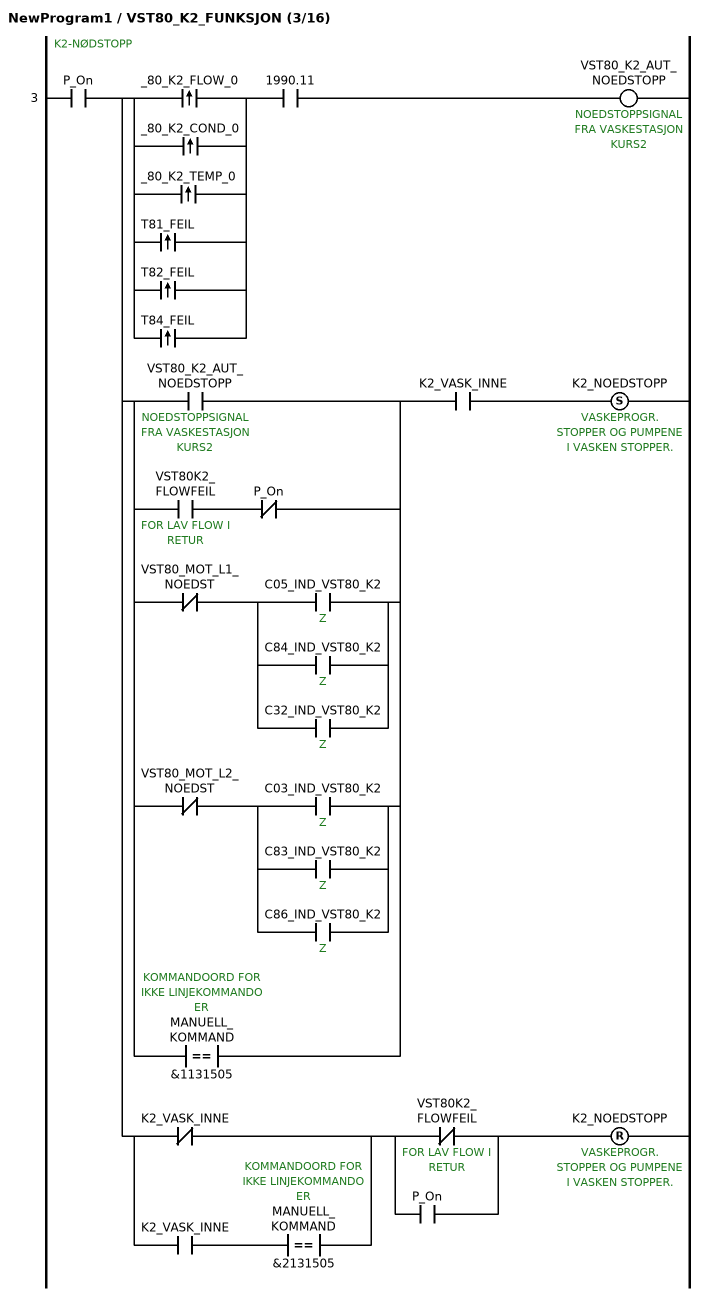
; rung 3: K2-NØDSTOPP
LD P_On
OUT TR0
@LD _80_K2_FLOW_0
@OR _80_K2_COND_0
@OR _80_K2_TEMP_0
@OR T81_FEIL
@OR T82_FEIL
@OR T84_FEIL
ANDLD
AND 1990.11
OUT VST80_K2_AUT_NOEDSTOPP  ; NOEDSTOPPSIGNAL FRA VASKESTASJON KURS2
LD TR0
LD VST80_K2_AUT_NOEDSTOPP  ; NOEDSTOPPSIGNAL FRA VASKESTASJON KURS2
LD VST80K2_FLOWFEIL  ; FOR LAV FLOW I RETUR
ANDNOT P_On
ORLD
LDNOT VST80_MOT_L1_NOEDST
LD C05_IND_VST80_K2  ; Z
OR C84_IND_VST80_K2  ; Z
OR C32_IND_VST80_K2  ; Z
ANDLD
ORLD
LDNOT VST80_MOT_L2_NOEDST
LD C03_IND_VST80_K2  ; Z
OR C83_IND_VST80_K2  ; Z
OR C86_IND_VST80_K2  ; Z
ANDLD
ORLD
OR=L(301) MANUELL_KOMMAND &1131505  ; KOMMANDOORD FOR IKKE LINJEKOMMANDOER
ANDLD
AND K2_VASK_INNE
SET K2_NOEDSTOPP  ; VASKEPROGR. STOPPER OG PUMPENE I VASKEN STOPPER.
LD TR0
LDNOT K2_VASK_INNE
LD K2_VASK_INNE
AND=L(301) MANUELL_KOMMAND &2131505  ; KOMMANDOORD FOR IKKE LINJEKOMMANDOER
ORLD
ANDLD
LDNOT VST80K2_FLOWFEIL  ; FOR LAV FLOW I RETUR
OR P_On
ANDLD
RSET K2_NOEDSTOPP  ; VASKEPROGR. STOPPER OG PUMPENE I VASKEN STOPPER.

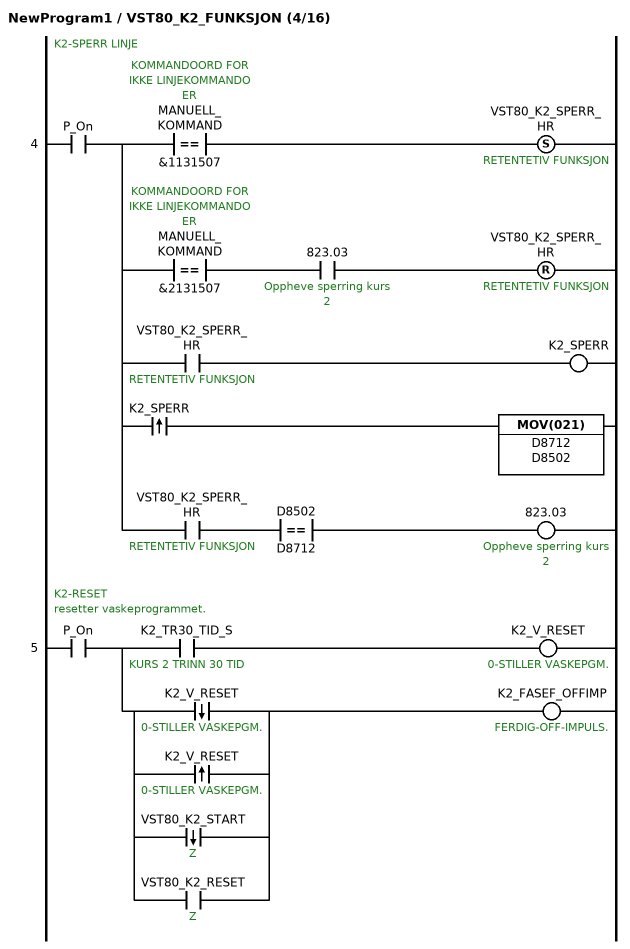
; rung 4: K2-SPERR LINJE
LD P_On
OUT TR0
AND=L(301) MANUELL_KOMMAND &1131507  ; KOMMANDOORD FOR IKKE LINJEKOMMANDOER
SET VST80_K2_SPERR_HR  ; RETENTETIV FUNKSJON
LD TR0
AND=L(301) MANUELL_KOMMAND &2131507  ; KOMMANDOORD FOR IKKE LINJEKOMMANDOER
AND 823.03  ; Oppheve sperring kurs 2
RSET VST80_K2_SPERR_HR  ; RETENTETIV FUNKSJON
LD TR0
AND VST80_K2_SPERR_HR  ; RETENTETIV FUNKSJON
OUT K2_SPERR
LD TR0
@AND K2_SPERR
MOV(021) D8712 D8502
LD TR0
AND VST80_K2_SPERR_HR  ; RETENTETIV FUNKSJON
AND=(300) D8502 D8712
OUT 823.03  ; Oppheve sperring kurs 2
; rung 5: K2-RESET / resetter vaskeprogrammet.
LD P_On
OUT TR0
AND K2_TR30_TID_S  ; KURS 2 TRINN 30 TID
OUT K2_V_RESET  ; 0-STILLER VASKEPGM.
LD TR0
%LD K2_V_RESET  ; 0-STILLER VASKEPGM.
@OR K2_V_RESET  ; 0-STILLER VASKEPGM.
%OR VST80_K2_START  ; Z
OR VST80_K2_RESET  ; Z
ANDLD
OUT K2_FASEF_OFFIMP  ; FERDIG-OFF-IMPULS.

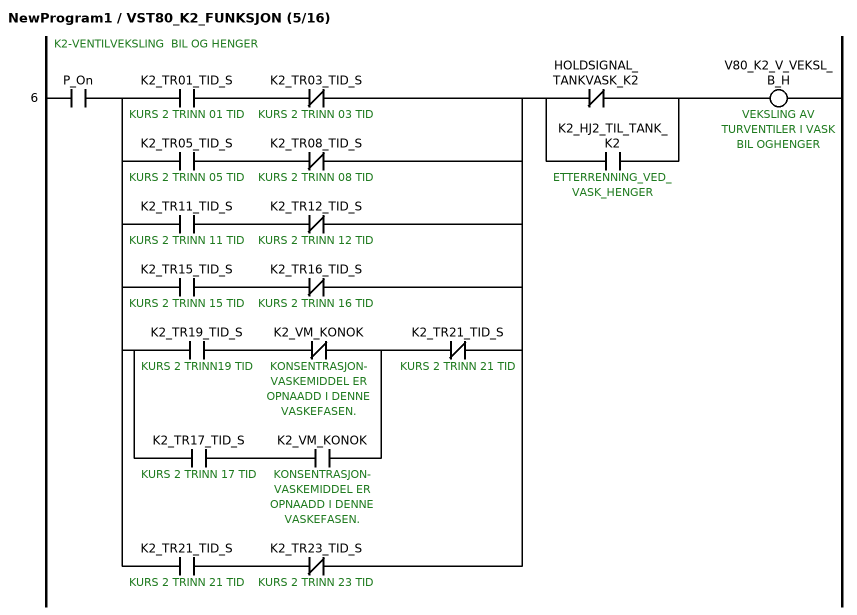
; rung 6: K2-VENTILVEKSLING  BIL OG HENGER
LD P_On
LD K2_TR01_TID_S  ; KURS 2 TRINN 01 TID
ANDNOT K2_TR03_TID_S  ; KURS 2 TRINN 03 TID
LD K2_TR05_TID_S  ; KURS 2 TRINN 05 TID
ANDNOT K2_TR08_TID_S  ; KURS 2 TRINN 08 TID
ORLD
LD K2_TR11_TID_S  ; KURS 2 TRINN 11 TID
ANDNOT K2_TR12_TID_S  ; KURS 2 TRINN 12 TID
ORLD
LD K2_TR15_TID_S  ; KURS 2 TRINN 15 TID
ANDNOT K2_TR16_TID_S  ; KURS 2 TRINN 16 TID
ORLD
LD K2_TR19_TID_S  ; KURS 2 TRINN19 TID
ANDNOT K2_VM_KONOK  ; KONSENTRASJON-VASKEMIDDEL ER OPNAADD I DENNE VASKEFASEN.
LD K2_TR17_TID_S  ; KURS 2 TRINN 17 TID
AND K2_VM_KONOK  ; KONSENTRASJON-VASKEMIDDEL ER OPNAADD I DENNE VASKEFASEN.
ORLD
ANDNOT K2_TR21_TID_S  ; KURS 2 TRINN 21 TID
ORLD
LD K2_TR21_TID_S  ; KURS 2 TRINN 21 TID
ANDNOT K2_TR23_TID_S  ; KURS 2 TRINN 23 TID
ORLD
ANDLD
LDNOT HOLDSIGNAL_TANKVASK_K2
OR K2_HJ2_TIL_TANK_K2  ; ETTERRENNING_VED_VASK_HENGER
ANDLD
OUT V80_K2_V_VEKSL_B_H  ; VEKSLING AV TURVENTILER I VASK BIL OGHENGER

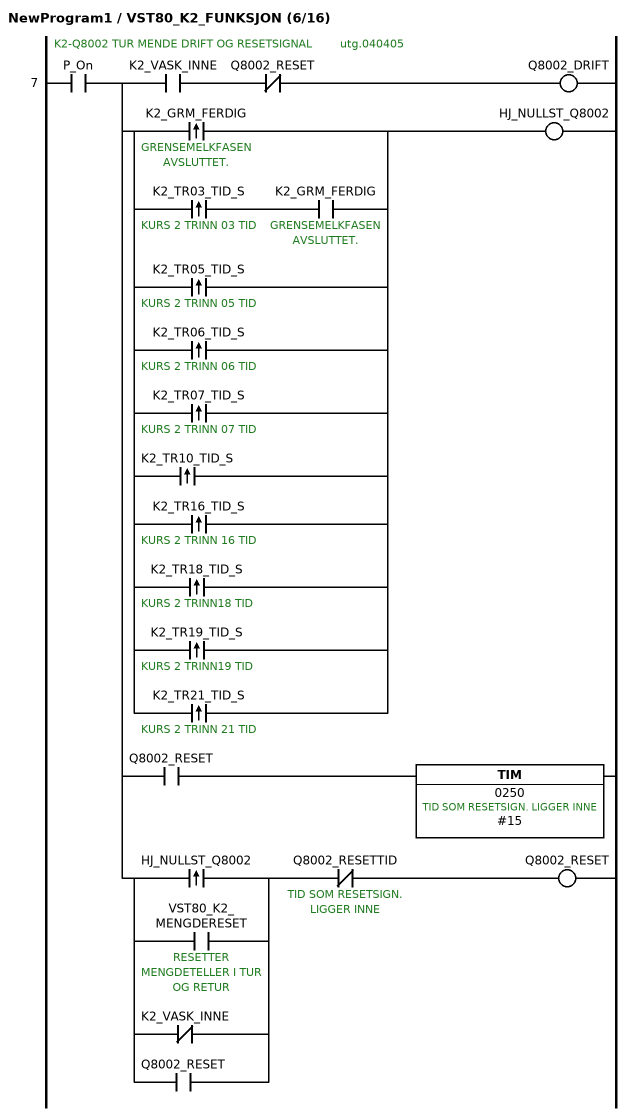
; rung 7: K2-Q8002 TUR MENDE DRIFT OG RESETSIGNAL        utg.040405
LD P_On
OUT TR0
AND K2_VASK_INNE
ANDNOT Q8002_RESET
OUT Q8002_DRIFT
LD TR0
@LD K2_GRM_FERDIG  ; GRENSEMELKFASEN AVSLUTTET.
@LD K2_TR03_TID_S  ; KURS 2 TRINN 03 TID
AND K2_GRM_FERDIG  ; GRENSEMELKFASEN AVSLUTTET.
ORLD
@OR K2_TR05_TID_S  ; KURS 2 TRINN 05 TID
@OR K2_TR06_TID_S  ; KURS 2 TRINN 06 TID
@OR K2_TR07_TID_S  ; KURS 2 TRINN 07 TID
@OR K2_TR10_TID_S
@OR K2_TR16_TID_S  ; KURS 2 TRINN 16 TID
@OR K2_TR18_TID_S  ; KURS 2 TRINN18 TID
@OR K2_TR19_TID_S  ; KURS 2 TRINN19 TID
@OR K2_TR21_TID_S  ; KURS 2 TRINN 21 TID
ANDLD
OUT HJ_NULLST_Q8002
LD TR0
AND Q8002_RESET
TIM 0250 #15  ; TID SOM RESETSIGN. LIGGER INNE
LD TR0
@LD HJ_NULLST_Q8002
OR VST80_K2_MENGDERESET  ; RESETTER MENGDETELLER I TUR OG RETUR
ORNOT K2_VASK_INNE
OR Q8002_RESET
ANDLD
ANDNOT Q8002_RESETTID  ; TID SOM RESETSIGN. LIGGER INNE
OUT Q8002_RESET

